FUNCTION F_StateValve_Process : bool
VAR_INPUT
END_VAR
VAR
END_VAR

F_StateValve_Process:= GVL_IO_VALVE.DO_00_V01ChalcogenCarrierChange = FALSE AND
				GVL_IO_VALVE.DO_00_V02MOCarreirChange = FALSE  AND
				GVL_IO_VALVE.DO_00_V03H2SeSourceChange = FALSE  AND
				GVL_IO_VALVE.DO_00_V04H2SSourceChange = FALSE ;

END_FUNCTION

(* stored: Version 1.1.0.1, ProductVersion 3.1.4024.15
   POU F_StateValve_Process: Id {d90acf08-ffd6-4205-a772-d8111e71dbdd}, SpecialFunc None *)
